# EPICS substitutions: iocBoot/iocxxx/examples/substitutions/AcsMotion_8.substitutions
#
# ACS Motion SPiiPlus motor substitutions for 8 axes
#
# Note: the P and PORT macros are passed from the dbLoadTemplate call.
# Edit the per-axis values (DESC, EGU, MRES, VELO, etc.) to match your hardware.
#

file "$(MOTOR)/db/asyn_motor.db"
{
pattern
{N,   M,       DTYP,         ADDR,  DESC,          EGU, DIR,  VELO,  VBAS,  ACCL,  BDST,  BVEL,  BACC,  MRES,      PREC,  DHLM,  DLLM,  INIT}
{1,  "m$(N)",  "asynMotor",  0,    "motor $(N)",  mm,  Pos,  1,     .1,    .2,    0,     1,     .2,    0.0001,    4,     100,   -100,  ""}
{2,  "m$(N)",  "asynMotor",  1,    "motor $(N)",  mm,  Pos,  1,     .1,    .2,    0,     1,     .2,    0.0001,    4,     100,   -100,  ""}
{3,  "m$(N)",  "asynMotor",  2,    "motor $(N)",  mm,  Pos,  1,     .1,    .2,    0,     1,     .2,    0.0001,    4,     100,   -100,  ""}
{4,  "m$(N)",  "asynMotor",  3,    "motor $(N)",  mm,  Pos,  1,     .1,    .2,    0,     1,     .2,    0.0001,    4,     100,   -100,  ""}
{5,  "m$(N)",  "asynMotor",  4,    "motor $(N)",  mm,  Pos,  1,     .1,    .2,    0,     1,     .2,    0.0001,    4,     100,   -100,  ""}
{6,  "m$(N)",  "asynMotor",  5,    "motor $(N)",  mm,  Pos,  1,     .1,    .2,    0,     1,     .2,    0.0001,    4,     100,   -100,  ""}
{7,  "m$(N)",  "asynMotor",  6,    "motor $(N)",  mm,  Pos,  1,     .1,    .2,    0,     1,     .2,    0.0001,    4,     100,   -100,  ""}
{8,  "m$(N)",  "asynMotor",  7,    "motor $(N)",  mm,  Pos,  1,     .1,    .2,    0,     1,     .2,    0.0001,    4,     100,   -100,  ""}
}

file "$(MOTOR)/db/profileMoveController.template"
{
pattern
{NAXES, NPOINTS, NPULSES, TIMEOUT}
{    8,    2000,    2000,     2.0}
}

file "$(MOTOR)/db/profileMoveAxis.template"
{
pattern
{M,   NPOINTS, NREADBACK, ADDR, TIMEOUT, PREC}
{1,     2000,      2000,  0,    2.0,    4}
{2,     2000,      2000,  1,    2.0,    4}
{3,     2000,      2000,  2,    2.0,    4}
{4,     2000,      2000,  3,    2.0,    4}
{5,     2000,      2000,  4,    2.0,    4}
{6,     2000,      2000,  5,    2.0,    4}
{7,     2000,      2000,  6,    2.0,    4}
{8,     2000,      2000,  7,    2.0,    4}
}

file "$(MOTOR)/db/SPiiPlusAxisExtra.db"
{
pattern
{M,    ADDR}
{m1,  0}
{m2,  1}
{m3,  2}
{m4,  3}
{m5,  4}
{m6,  5}
{m7,  6}
{m8,  7}
}

file "$(MOTOR)/db/SPiiPlusHoming.db"
{
pattern
{M,    ADDR, TIMEOUT,  VAL,  MAX_DIST, OFFSET_POS, OFFSET_NEG}
{m1,  0,    2.0,    0,    0.0,      0.0,        0.0}
{m2,  1,    2.0,    0,    0.0,      0.0,        0.0}
{m3,  2,    2.0,    0,    0.0,      0.0,        0.0}
{m4,  3,    2.0,    0,    0.0,      0.0,        0.0}
{m5,  4,    2.0,    0,    0.0,      0.0,        0.0}
{m6,  5,    2.0,    0,    0.0,      0.0,        0.0}
{m7,  6,    2.0,    0,    0.0,      0.0,        0.0}
{m8,  7,    2.0,    0,    0.0,      0.0,        0.0}
}

file "$(MOTOR)/db/SPiiPlusJogging.db"
{
pattern
{M}
{m1}
{m2}
{m3}
{m4}
{m5}
{m6}
{m7}
{m8}
}

# Customize MAX_VELO and MAX_ACCL per motor as needed
file "$(MOTOR)/db/SPiiPlusMaxParams.db"
{
pattern
{M,    ADDR,  MAX_VELO,  MAX_ACCL,  PREC}
{m1,  0,       5.0,      20.0,     4}
{m2,  1,       5.0,      20.0,     4}
{m3,  2,       5.0,      20.0,     4}
{m4,  3,       5.0,      20.0,     4}
{m5,  4,       5.0,      20.0,     4}
{m6,  5,     200.0,    1000.0,     4}
{m7,  6,     200.0,    1000.0,     4}
{m8,  7,     200.0,    1000.0,     4}
}

file "$(MOTOR)/db/SPiiPlusMaxParamsRbv.db"
{
pattern
{M,    ADDR, PREC}
{m1,  0,   4}
{m2,  1,   4}
{m3,  2,   4}
{m4,  3,   4}
{m5,  4,   4}
{m6,  5,   4}
{m7,  6,   4}
{m8,  7,   4}
}

### The feedback database is helpful for troubleshooting encoder problems
file "$(MOTOR)/db/SPiiPlusFeedback.db"
{
pattern
{M,    ADDR, PREC, SCAN}
{m1,  0,   6,    2}
{m2,  1,   6,    2}
{m3,  2,   6,    2}
{m4,  3,   6,    2}
{m5,  4,   6,    2}
{m6,  5,   6,    2}
{m7,  6,   6,    2}
{m8,  7,   6,    2}
}
